FUNCTION_BLOCK SKILL_Core (* Skill core: state machine, OPC UA Stop/Abort/Reset(Session) -> [Accepted, ErrorID], State and ErrorID published, activity counted; the Start method (with the skill's parameters) is wired to CMD_START and RSP_START; GO starts the execution, SUCCESS or FAILURE(ErrorID) ends it *)
  (* Standard: 61499-2 *)
  (* Version 0.1, 2026-09-28, Project contributors, AAU Smart Production Lab *)
  PACKAGE modlib;
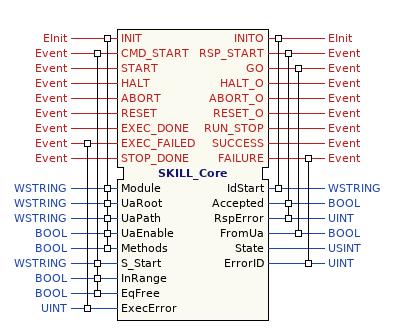
  EVENT_INPUT
    INIT : EInit WITH Module, UaRoot, UaPath, UaEnable, Methods;
    CMD_START WITH S_Start, InRange, EqFree;
    START;
    HALT;
    ABORT;
    RESET;
    EXEC_DONE;
    EXEC_FAILED WITH ExecError;
    STOP_DONE;
  END_EVENT
  EVENT_OUTPUT
    INITO : EInit WITH IdStart;
    RSP_START WITH Accepted, RspError;
    GO WITH FromUa;
    HALT_O;
    ABORT_O;
    RESET_O;
    RUN_STOP;
    SUCCESS;
    FAILURE WITH ErrorID;
  END_EVENT
  VAR_INPUT
    Module : WSTRING;
    UaRoot : WSTRING;
    UaPath : WSTRING;
    UaEnable : BOOL;
    Methods : BOOL;
    S_Start : WSTRING;
    InRange : BOOL := TRUE;
    EqFree : BOOL := TRUE;
    ExecError : UINT;
  END_VAR
  VAR_OUTPUT
    IdStart : WSTRING;
    Accepted : BOOL;
    RspError : UINT;
    FromUa : BOOL;
    State : USINT;
    ErrorID : UINT;
  END_VAR
  FBS
    Control : modlib::SKILL_Control;
    Owner : modlib::MOD_OwnerView;
    Mode : modlib::MOD_StateView;
    UaStop : iec61499::net::SERVER_2_1;
    UaAbort : iec61499::net::SERVER_2_1;
    UaReset : iec61499::net::SERVER_2_1;
    PubState : iec61499::net::PUBLISH_2;
    Act : iec61499::net::PUBLISH_1(QI := TRUE);
    ToIdle : iec61499::events::E_DELAY(DT := T#1500ms);
  END_FBS
  EVENT_CONNECTIONS
    INIT TO Control.INIT;
    Control.INITO TO Owner.INIT;
    Owner.INITO TO Mode.INIT;
    Mode.INITO TO UaStop.INIT;
    UaStop.INITO TO UaAbort.INIT;
    UaAbort.INITO TO UaReset.INIT;
    UaReset.INITO TO PubState.INIT;
    PubState.INITO TO Act.INIT;
    Act.INITO TO PubState.REQ;
    Act.INITO TO INITO;
    CMD_START TO Control.CMD_START;
    Control.RSP_START TO RSP_START;
    UaStop.IND TO Control.CMD_STOP;
    Control.RSP_STOP TO UaStop.RSP;
    UaAbort.IND TO Control.CMD_ABORT;
    Control.RSP_ABORT TO UaAbort.RSP;
    UaReset.IND TO Control.CMD_RESET;
    Control.RSP_RESET TO UaReset.RSP;
    Owner.CHG TO Control.OWNER_CHG;
    Mode.CHG TO Control.MOD_CHG;
    Control.PUB TO PubState.REQ;
    Control.ACT TO Act.REQ;
    START TO Control.START;
    HALT TO Control.HALT;
    ABORT TO Control.ABORT;
    RESET TO Control.RESET;
    EXEC_DONE TO Control.EXEC_DONE;
    EXEC_FAILED TO Control.EXEC_FAILED;
    STOP_DONE TO Control.STOP_DONE;
    Control.GO TO GO;
    Control.HALT_O TO HALT_O;
    Control.ABORT_O TO ABORT_O;
    Control.RESET_O TO RESET_O;
    Control.RUN_STOP TO RUN_STOP;
    Control.SUCCESS TO SUCCESS;
    Control.FAILURE TO FAILURE;
    Control.TO_IDLE_START TO ToIdle.START;
    Control.TO_IDLE_STOP TO ToIdle.STOP;
    ToIdle.EO TO Control.TO_IDLE;
  END_CONNECTIONS
  DATA_CONNECTIONS
    Module TO Control.Module;
    Module TO Owner.Module;
    Module TO Mode.Module;
    UaRoot TO Control.UaRoot;
    UaPath TO Control.UaPath;
    Methods TO UaStop.QI;
    Methods TO UaAbort.QI;
    Methods TO UaReset.QI;
    UaEnable TO PubState.QI;
    Control.IdStart TO IdStart;
    S_Start TO Control.S_Start;
    InRange TO Control.InRange;
    EqFree TO Control.EqFree;
    Control.Accepted TO Accepted;
    Control.Accepted TO UaStop.SD_1;
    Control.Accepted TO UaAbort.SD_1;
    Control.Accepted TO UaReset.SD_1;
    Control.RspError TO RspError;
    Control.RspError TO UaStop.SD_2;
    Control.RspError TO UaAbort.SD_2;
    Control.RspError TO UaReset.SD_2;
    Control.IdStop TO UaStop.ID;
    UaStop.RD_1 TO Control.S_Stop;
    Control.IdAbort TO UaAbort.ID;
    UaAbort.RD_1 TO Control.S_Abort;
    Control.IdReset TO UaReset.ID;
    UaReset.RD_1 TO Control.S_Reset;
    Owner.Owner TO Control.Owner;
    Mode.State TO Control.ModState;
    Control.IdPub TO PubState.ID;
    Control.State TO PubState.SD_1;
    Control.State TO State;
    Control.ErrorID TO PubState.SD_2;
    Control.ErrorID TO ErrorID;
    Control.IdAct TO Act.ID;
    Control.Delta TO Act.SD_1;
    ExecError TO Control.ExecError;
    Control.FromUa TO FromUa;
  END_CONNECTIONS
END_FUNCTION_BLOCK
